FUNCTION_BLOCK FB_pushBtnNC
VAR
	bBtn AT %I* : BOOL;
END_VAR

PROPERTY isPressed : BOOL
GET
IF NOT bBtn THEN 
	isPressed := TRUE;
ELSE 
	isPressed := FALSE;
END_IF
END_GET
END_PROPERTY

END_FUNCTION_BLOCK

(* stored: Version 1.1.0.1, ProductVersion 3.1.4024.13
   POU FB_pushBtnNC: Id {26c5556c-fe5e-424d-a946-f4ffef02553f}, SpecialFunc None
   Property isPressed: Id {ffc4e911-297d-4446-b02b-a64e5fc500ba}
   Get Get: Id {37011f4a-2da0-488f-916f-a5b833c89d0a} *)
